PROGRAM MAIN
VAR
	ready				: BOOL;		// telescope drives are ready to enable
	error				: BOOL;
	brakeClearing		: BOOL := FALSE;	//	open brake
	
	commTimer 			: TON := (PT:=T#5S);
	getHostName			: FB_GetHostName;
	hostName			: STRING(255);
	executeHostName		: BOOL := TRUE;
	
	eTelescopeMode 		: E_TelescopeMode;
	
	fbComm				: FB_Comm_MQTT_Influx;
	SafetyHandling		: FB_MonetSafetyHandling(comm := fbComm);
	CabinetControl		: FB_MonetCabinetControl(comm := fbComm);
	PowerMonitoring		: FB_MonetPowerMonitoring(comm := fbComm);
	RoofControl			: FB_RoofControl(comm := fbComm);
	CoverControl		: FB_MonetCoverControl(comm := fbComm);
	HydraulicsControl	: FB_HydraulicsControl(comm := fbComm);
	FocusControl		: FB_FocusControl(comm := fbComm);
	DerotatorControl	: FB_DerotatorControl(comm := fbComm);
	ElevationControl	: FB_ElevationControl(comm := fbComm);
	AzimuthControl		: FB_AzimuthControl(comm := fbComm);
	TelescopeControl	: FB_MonetTelescopeControl(comm := fbComm);
	TelescopeAuxiliary  : FB_TelescopeAuxiliary(comm := fbComm);
	PendantControl		: FB_MonetPendantControl(comm := fbComm);
	
	//fbWeather			: FB_WeatherCheck();
	
	MqttWatchdog		: FB_MonetMqttWatchdog(comm := fbComm);	// park + close roof after 30 s without broker (MONETcommon)
	Diagnostics			: FB_MonetDiagnostics(comm := fbComm);	// diagnostics/base/* telemetry, on change + 30 s heartbeat (MONETcommon)
END_VAR
VAR CONSTANT
	telescopeConfig		: ST_TelescopeConfig := (longitude := 20.810808, latitude := -32.375823, altitude := 1798.0, 
												 azimuthPark := 175, elevationPark := 60, derotatorPark := 0, focusPark := 36.0, 
												 azimuthHome := 175, elevationHome := 40, derotatorHome := 0,
												 name := 'MONET/S', diameter := 1.2, cabinet := 'Beckhoff', manufacturer := 'Halfmann, Haidenhain, Beckhoff',
												 mountOptions := 'ALT-AZ', mount := 'ALT_AZ');
	fbPointing			: FB_PointingModelForward(AOFF := -0.006778523308102358, BNP := 0.030459575443670728, AN_A := -0.013961935190411667, AE_A := -0.01036163798027645, NPAE := 0.0017131069293910839, 
                                                  EOFF := 0.04040337399598415, AN_E := -0.011190631316106092, AE_E := -0.009741636951375865, TF := 0.06450337748465318);
	fbPointingInverse	: FB_PointingModelInversion(fbPointing := fbPointing);
END_VAR

(* 
Main control loop
* Execute sub modules
* power management
* control panel switches and status lamps

* start switch activates Hydraulics and Trafo
* 
*)

// get hostname for MQTT connection
GetHostName(bExecute := executeHostName, sHostName => HostName);
executeHostName := FALSE;

// run cabinet
CabinetControl();

// telescope mode
IF CabinetControl.KeyLocal THEN
	eTelescopeMode := SEL(HydraulicsControl.Enable, E_TelescopeMode.off, E_TelescopeMode.manual);	
ELSE
	eTelescopeMode := E_TelescopeMode.automatic; 
END_IF

// in local mode we can start or stop hydraulics and open the brake
brakeClearing := TRUE;
IF eTelescopeMode = E_TelescopeMode.manual OR eTelescopeMode = E_TelescopeMode.off THEN
	IF CabinetControl.IsStartPushed() THEN
		HydraulicsControl.Enable := TRUE;
	END_IF
	IF CabinetControl.IsStopPushed() THEN
		HydraulicsControl.Enable := FALSE;
	END_IF
	brakeClearing := CabinetControl.AreBreakesCleared();
	HydraulicsControl.bOpenBrake := brakeClearing;
END_IF

// clear errors: SafetyHandling.resetRequest (see call below) toggles Restart/ErrAck,
// here the cabinet/pendant reset button also resets covers, hydraulics and, in automatic mode, the
// telescope control (the only way to clear a latched bInterrupted)
IF CabinetControl.IsResetPushed() OR PendantControl.IbResetButton THEN
	CoverControl.Reset();
	HydraulicsControl.Reset();
	IF eTelescopeMode = E_TelescopeMode.automatic THEN
		TelescopeControl.Reset();
	END_IF
END_IF

// telescope is ready when power available
PowerMonitoring(phaseOK => ready);

// only run TelescopeControl in automatic mode
IF eTelescopeMode = E_TelescopeMode.automatic THEN
	TelescopeControl(
		telescopeConfig := telescopeConfig,
		fbCovers 		:= CoverControl,
		fbBrake 		:= HydraulicsControl,
		fbHydraulics 	:= HydraulicsControl,
		fbFocus 		:= FocusControl,
		fbElevation 	:= ElevationControl,
		fbAzimuth 		:= AzimuthControl,
		fbDerotator 	:= DerotatorControl,
		fbPointing      := fbPointing,
		fbPointingInverse := fbPointingInverse,
		bEstopTriggered := SafetyHandling.estop,	// M5: was never wired, see MONETcommon#11
		bMainReady		:= ready					// M5: was computed and published but never wired, see MONETcommon#11
	);
END_IF
TelescopeAuxiliary();

// run all control FBs
CoverControl();
HydraulicsControl(
	nMinPanLevel	:= 3500,
	nMaxPanLevel	:= 10200,
	fMinPanPercent	:= 0.0,
	fMaxPanPercent	:= 50.0, //56.0,
	bBrakeClearing	:= brakeClearing
);
ElevationControl(
	fCalibPosition 	:= 60.567917554230512,
	fbCovers 		:= CoverControl, 
	fbBrake 		:= HydraulicsControl
);
AzimuthControl(
	fCalibPosition	:= 1.1466144421902693,
	fMinPosition	:= -274.0,
	fMaxPosition	:= 270.0,
	bBrakeOpen		:= HydraulicsControl.brakeOpen,
);
DerotatorControl(
	fMinPosition		:= -90.0,
	fMaxPosition		:= 360.0
);	//
FocusControl(
	eTelescopeMode 	:= eTelescopeMode,
	fHomingPosition	:= 92.02, // 104.02 - 12.00
	fVelocity		:= 0.2,
	ptBrakeDelay	:= T#30S,
	ptFocusDelay	:= T#100MS
);
RoofControl(
	min_speed		:= 10000,
	max_speed 		:= 30000, 
	acceleration 	:= 150,
	max_position_1 	:= 205,
	max_position_2 	:= 203,
	max_position_diff	:= 3,
	limit_slowdown	:= 5
);
PendantControl(
	fbCovers 		:= CoverControl, 
	fbBrake 		:= HydraulicsControl, 
	fbHydraulics 	:= HydraulicsControl, 
	fbFocus 		:= FocusControl, 
	fbElevation 	:= ElevationControl, 
	fbAzimuth 		:= AzimuthControl, 
	fbDerotator 	:= DerotatorControl	
);

// MQTT watchdog: if connection is lost for more than the timeout, park and close roof.
// Armed only after the first successful connect -- otherwise a normal boot (bConnected
// starts FALSE until the initial hostname/connect/subscribe sequence completes) would
// trip this on every restart, not just real outages.
MqttWatchdog(bConnected := fbComm.bConnected, iTelescope := TelescopeControl, iRoof := RoofControl);

// and fbComm
fbComm(	
	sHostName		:= '192.168.127.10',
    nHostPort  		:= 1883,
    nKeepAlive  	:= 60,
	sTopicSub  		:= 'MONETS/Telescope/SET',
	sTopicPublish	:= 'MONETS/Telemetry',
	sTopicLog		:= 'MONETS/Log',
	Telescope		:= TelescopeControl,
	AltAzTelescope  := TelescopeControl,
	Focus			:= FocusControl,
	Roof			:= RoofControl
);

// check weather and UPSs
//fbWeather(
//	sHostName		:= '192.168.127.10',
//	nHostPort       := 8002,
//	sUri			:= '/api/current/'
//);
//IF fbWeather.bError OR NOT fbWeather.bWeatherGood THEN
	//TelescopeControl.Park();
	//RoofControl.Close();
//END_IF

// set control lights
//error := Focuscontrol.Error OR CoverControl.Error OR HydraulicsControl.Error;
error := CoverControl.Error OR HydraulicsControl.Error;
CabinetControl.SetManualLamp(eTelescopeMode = E_TelescopeMode.manual);

// blink errors
IF SafetyHandling.error THEN
	CabinetControl.SetBlinkError(E_Blink.short);
ELSIF ElevationControl.bError OR AzimuthControl.bError OR DerotatorControl.bError THEN
	CabinetControl.SetBlinkError(E_Blink.long);
ELSIF HydraulicsControl.bOilWarning OR HydraulicsControl.bOilHot OR HydraulicsControl.bPressureFailure THEN
	CabinetControl.SetBlinkError(E_Blink.slow);
ELSIF error THEN
	CabinetControl.SetBlinkError(E_Blink.on);
ELSE
	CabinetControl.SetBlinkError(E_Blink.off); 
END_IF

// power lamp is always on
CabinetControl.SetBlinkPower(E_Blink.on);

// do safety
SafetyHandling(resetRequest := CabinetControl.IsResetPushed() OR PendantControl.IbResetButton);

// telemetry
commTimer(IN:=TRUE);
IF commTimer.Q THEN
	commTimer(IN:=FALSE);
	fbComm.Publish('electronics', 'base', 'MainReady', BOOL_TO_STRING(ready));
	fbComm.Publish('electronics', 'base', 'MasterError', BOOL_TO_STRING(error));
	TelescopeAuxiliary.SendTelemetry();
END_IF

// diagnostics telemetry: publish on change, plus a full-snapshot heartbeat (MONETcommon)
Diagnostics(
	fbTelescope	:= TelescopeControl,
	fbElevation	:= ElevationControl,
	fbAzimuth	:= AzimuthControl,
	fbDerotator	:= DerotatorControl,
	fbFocus		:= FocusControl,
	fbSafety	:= SafetyHandling
);

END_PROGRAM

(* stored: Version 1.1.0.1, ProductVersion 3.1.4024.15
   POU MAIN: Id {0fe844df-7078-44d3-bc48-268e6c994874}, SpecialFunc None *)
